Fanuc KAREL source: CNC_DYN_DISI.kl

PROGRAM T
%NOLOCKGROUP
VAR
 v0 : INTEGER
 v1 : STRING[40]
 v2 : INTEGER
BEGIN
 CNC_DYN_DISI(v0, v1, v2)
END T
